PROGRAM V0_5
VAR
END_VAR

(*
	Opslagvat met foutdetectie
	
	In de voorgaande oefening werden twee sensoren voor niveaudetectie gebruikt. Het is onmogelijk dat de sensor onderaan geen vloeistof detecteert (FALSE)
	en de sensor bovenaan de tank wel (TRUE). De sensor onderaan moet dus defect zijn of er is een kabelbreuk. In dat geval mogen noch de klep, noch de pomp geactiveerd kunnen worden.
	
	bSwitch_1 = Hoog niveau (L1)
	bSwitch_2 = Laag niveau (L2)
	bLamp_1 = Klep (K1)
	bLamp_2 = Pomp (P1)
	bButton_1 = Pomp start (B1)
	bButton_2 = Pomp stop (B2)
	
	(T = Toggle)
	L1	l2	B1	B2	P1	K1
	0	0	x	x	x	1	-- Sturing klep
	1	0	x	x	x	0
	1	1	x	x	x	0
	0	1	x	x	x	1
	
	x	1	1	0	1	x	-- Sturing pomp
	x	1	0	1	0	x
	x	0	x	x	0	x	
*)

// Sturing klep
GVL.bLamp_1 := (NOT GVL.bSwitch_1 AND NOT GVL.bSwitch_2) OR (NOT GVL.bSwitch_1 AND GVL.bSwitch_2);

// Sturing pomp
GVL.bLamp_2 S= GVL.bSwitch_2 AND GVL.bButton_1;
GVL.bLamp_2 R= (GVL.bSwitch_2 AND GVL.bButton_2) OR (GVL.bSwitch_1 AND NOT GVL.bSwitch_2) OR NOT GVL.bSwitch_2;

END_PROGRAM

(* stored: Version 1.1.0.1, ProductVersion 3.1.4024.12
   POU V0_5: Id {2b831544-7a60-4222-bc09-e5d3f07db049}, SpecialFunc None *)
